// TIA Portal V16 export
// export: Created 2021-11-12T13:32:07.3551266Z, ExportSetting WithDefaults, DisplayName Totally Integrated Automation Portal, DisplayVersion V16 Update 3, DisplayName TIA Portal Version Control Interface, DisplayVersion V16 Update 2, DisplayName TIA Portal Openness, DisplayVersion V16 Update 3, DisplayName SINAMICS Startdrive Advanced, DisplayVersion V16 Update 5, DisplayName SINAMICS Startdrive G130, G150, S120, S150, SINAMICS MV, S210, DisplayVersion V16 Update 5, DisplayName SINAMICS Startdrive G110M, G120, G120C, G120D, G120P, G115D, DisplayVersion V16 Update 5, DisplayName STEP 7 Professional, DisplayVersion V16 Update 3, DisplayName STEP 7 Safety, DisplayVersion V16, DisplayName WinCC UA Professional, DisplayVersion V16 Update 3
FUNCTION_BLOCK "Station130"   // FB11, LAD
{ S7_Optimized_Access := 'TRUE' }
VERSION : 0.1
// stored: AutoNumber true, IsIECCheckEnabled false, IsRetainMemResEnabled false, MemoryReserve 100, SetENOAutomatically false, UDAEnableTagReadback false
   VAR
      SS_RobotZones : "STD_RobotZones";
      SI_PartType { S7_SetPoint := 'True'} : Int;
      SDI_PartID : DInt;
      SI_PartCounter : Int;
   END_VAR
   VAR_TEMP   // added for the SCL form of the ladder/FBD networks
      _w1 : Bool;
      _w2 : Bool;
      _w3 : Bool;
      _w4 : Bool;
      _w5 : Bool;
      _w6 : Bool;
      _w7 : Bool;
      _w8 : Bool;
      _w9 : Bool;
      _w10 : Bool;
      _w11 : Bool;
      _w12 : Bool;
      _w13 : Bool;
      _w14 : Bool;
      _w15 : Bool;
      _w16 : Bool;
      _w17 : Bool;
      _w18 : Bool;
      _w19 : Bool;
      _w20 : Bool;
      _w21 : Bool;
      _w22 : Bool;
      _w23 : Bool;
      _w24 : Bool;
      _w25 : Bool;
   END_VAR
BEGIN

REGION Network 1: *************** Clear Temporary ***************
END_REGION

REGION Network 2: *************** Zone release *************
END_REGION

REGION Network 3: Enable for robots 1R1, 1R3 to enter zone 130
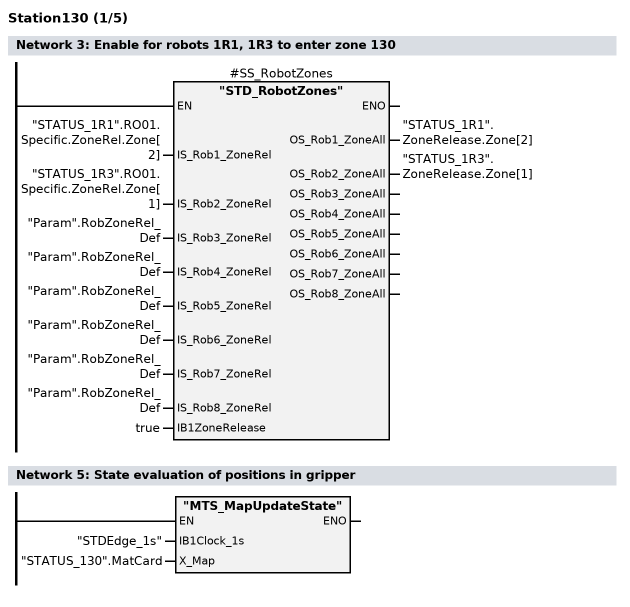
   RUNG wire#powerrail
      #SS_RobotZones(IS_Rob1_ZoneRel := "STATUS_1R1".RO01.Specific.ZoneRel.Zone[2], IS_Rob2_ZoneRel := "STATUS_1R3".RO01.Specific.ZoneRel.Zone[1], IS_Rob3_ZoneRel := "Param".RobZoneRel_Def, IS_Rob4_ZoneRel := "Param".RobZoneRel_Def, IS_Rob5_ZoneRel := "Param".RobZoneRel_Def, IS_Rob6_ZoneRel := "Param".RobZoneRel_Def, IS_Rob7_ZoneRel := "Param".RobZoneRel_Def, IS_Rob8_ZoneRel := "Param".RobZoneRel_Def, IB1ZoneRelease := true, OS_Rob1_ZoneAll => "STATUS_1R1".ZoneRelease.Zone[2], OS_Rob2_ZoneAll => "STATUS_1R3".ZoneRelease.Zone[1], OS_Rob3_ZoneAll =>, OS_Rob4_ZoneAll =>, OS_Rob5_ZoneAll =>, OS_Rob6_ZoneAll =>, OS_Rob7_ZoneAll =>, OS_Rob8_ZoneAll =>)
   END_RUNG
   // the same network as SCL:
   #SS_RobotZones(IS_Rob1_ZoneRel := "STATUS_1R1".RO01.Specific.ZoneRel.Zone[2],   // "STD_RobotZones"
                  IS_Rob2_ZoneRel := "STATUS_1R3".RO01.Specific.ZoneRel.Zone[1],
                  IS_Rob3_ZoneRel := "Param".RobZoneRel_Def,
                  IS_Rob4_ZoneRel := "Param".RobZoneRel_Def,
                  IS_Rob5_ZoneRel := "Param".RobZoneRel_Def,
                  IS_Rob6_ZoneRel := "Param".RobZoneRel_Def,
                  IS_Rob7_ZoneRel := "Param".RobZoneRel_Def,
                  IS_Rob8_ZoneRel := "Param".RobZoneRel_Def,
                  IB1ZoneRelease := true,
                  OS_Rob1_ZoneAll => "STATUS_1R1".ZoneRelease.Zone[2],
                  OS_Rob2_ZoneAll => "STATUS_1R3".ZoneRelease.Zone[1]);
END_REGION

REGION Network 4: *************** Material flow ***************
END_REGION

REGION Network 5: State evaluation of positions in gripper
   RUNG wire#powerrail
      "MTS_MapUpdateState"(IB1Clock_1s := "STDEdge_1s", X_Map := "STATUS_130".MatCard)
   END_RUNG
   // the same network as SCL:
   "MTS_MapUpdateState"(IB1Clock_1s := "STDEdge_1s", X_Map := "STATUS_130".MatCard);
END_REGION

REGION Network 6: Clear positions and map - commands
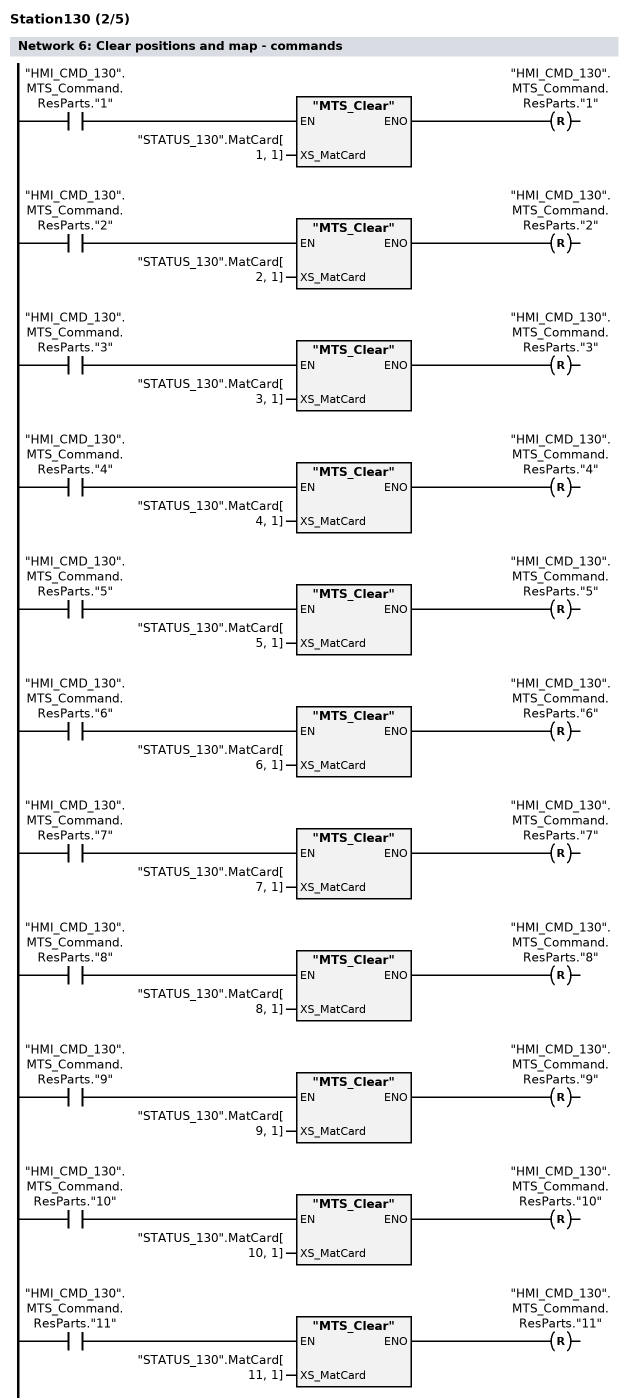
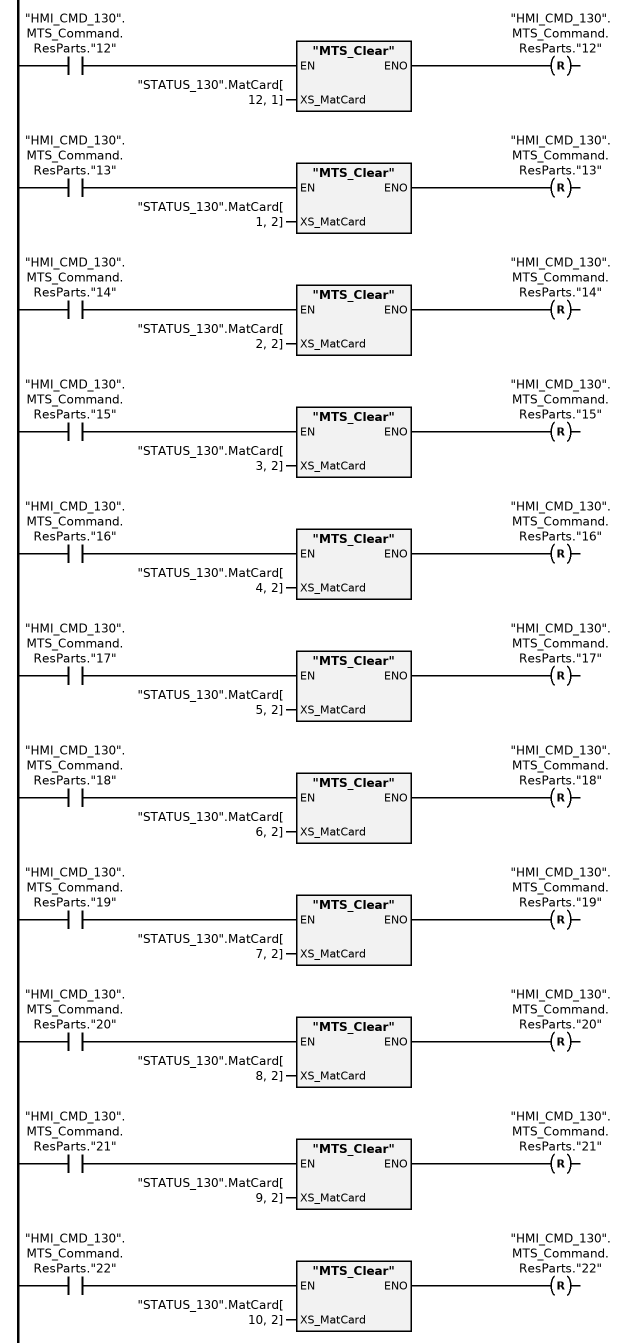
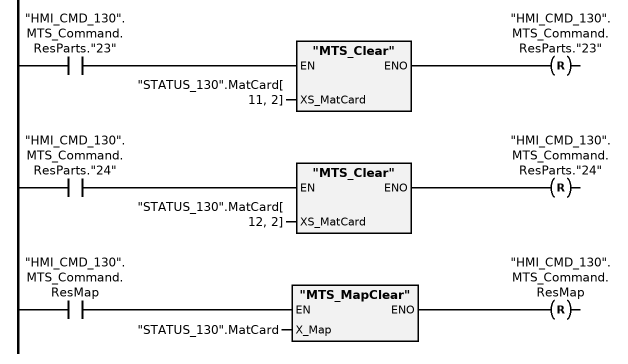
   RUNG wire#powerrail
      Contact( "HMI_CMD_130".MTS_Command.ResParts."1" )
      "MTS_Clear"(XS_MatCard := "STATUS_130".MatCard[1, 1])
      R_Coil( "HMI_CMD_130".MTS_Command.ResParts."1" )
   END_RUNG
   RUNG wire#powerrail
      Contact( "HMI_CMD_130".MTS_Command.ResParts."2" )
      "MTS_Clear"(XS_MatCard := "STATUS_130".MatCard[2, 1])
      R_Coil( "HMI_CMD_130".MTS_Command.ResParts."2" )
   END_RUNG
   RUNG wire#powerrail
      Contact( "HMI_CMD_130".MTS_Command.ResParts."3" )
      "MTS_Clear"(XS_MatCard := "STATUS_130".MatCard[3, 1])
      R_Coil( "HMI_CMD_130".MTS_Command.ResParts."3" )
   END_RUNG
   RUNG wire#powerrail
      Contact( "HMI_CMD_130".MTS_Command.ResParts."4" )
      "MTS_Clear"(XS_MatCard := "STATUS_130".MatCard[4, 1])
      R_Coil( "HMI_CMD_130".MTS_Command.ResParts."4" )
   END_RUNG
   RUNG wire#powerrail
      Contact( "HMI_CMD_130".MTS_Command.ResParts."5" )
      "MTS_Clear"(XS_MatCard := "STATUS_130".MatCard[5, 1])
      R_Coil( "HMI_CMD_130".MTS_Command.ResParts."5" )
   END_RUNG
   RUNG wire#powerrail
      Contact( "HMI_CMD_130".MTS_Command.ResParts."6" )
      "MTS_Clear"(XS_MatCard := "STATUS_130".MatCard[6, 1])
      R_Coil( "HMI_CMD_130".MTS_Command.ResParts."6" )
   END_RUNG
   RUNG wire#powerrail
      Contact( "HMI_CMD_130".MTS_Command.ResParts."7" )
      "MTS_Clear"(XS_MatCard := "STATUS_130".MatCard[7, 1])
      R_Coil( "HMI_CMD_130".MTS_Command.ResParts."7" )
   END_RUNG
   RUNG wire#powerrail
      Contact( "HMI_CMD_130".MTS_Command.ResParts."8" )
      "MTS_Clear"(XS_MatCard := "STATUS_130".MatCard[8, 1])
      R_Coil( "HMI_CMD_130".MTS_Command.ResParts."8" )
   END_RUNG
   RUNG wire#powerrail
      Contact( "HMI_CMD_130".MTS_Command.ResParts."9" )
      "MTS_Clear"(XS_MatCard := "STATUS_130".MatCard[9, 1])
      R_Coil( "HMI_CMD_130".MTS_Command.ResParts."9" )
   END_RUNG
   RUNG wire#powerrail
      Contact( "HMI_CMD_130".MTS_Command.ResParts."10" )
      "MTS_Clear"(XS_MatCard := "STATUS_130".MatCard[10, 1])
      R_Coil( "HMI_CMD_130".MTS_Command.ResParts."10" )
   END_RUNG
   RUNG wire#powerrail
      Contact( "HMI_CMD_130".MTS_Command.ResParts."11" )
      "MTS_Clear"(XS_MatCard := "STATUS_130".MatCard[11, 1])
      R_Coil( "HMI_CMD_130".MTS_Command.ResParts."11" )
   END_RUNG
   RUNG wire#powerrail
      Contact( "HMI_CMD_130".MTS_Command.ResParts."12" )
      "MTS_Clear"(XS_MatCard := "STATUS_130".MatCard[12, 1])
      R_Coil( "HMI_CMD_130".MTS_Command.ResParts."12" )
   END_RUNG
   RUNG wire#powerrail
      Contact( "HMI_CMD_130".MTS_Command.ResParts."13" )
      "MTS_Clear"(XS_MatCard := "STATUS_130".MatCard[1, 2])
      R_Coil( "HMI_CMD_130".MTS_Command.ResParts."13" )
   END_RUNG
   RUNG wire#powerrail
      Contact( "HMI_CMD_130".MTS_Command.ResParts."14" )
      "MTS_Clear"(XS_MatCard := "STATUS_130".MatCard[2, 2])
      R_Coil( "HMI_CMD_130".MTS_Command.ResParts."14" )
   END_RUNG
   RUNG wire#powerrail
      Contact( "HMI_CMD_130".MTS_Command.ResParts."15" )
      "MTS_Clear"(XS_MatCard := "STATUS_130".MatCard[3, 2])
      R_Coil( "HMI_CMD_130".MTS_Command.ResParts."15" )
   END_RUNG
   RUNG wire#powerrail
      Contact( "HMI_CMD_130".MTS_Command.ResParts."16" )
      "MTS_Clear"(XS_MatCard := "STATUS_130".MatCard[4, 2])
      R_Coil( "HMI_CMD_130".MTS_Command.ResParts."16" )
   END_RUNG
   RUNG wire#powerrail
      Contact( "HMI_CMD_130".MTS_Command.ResParts."17" )
      "MTS_Clear"(XS_MatCard := "STATUS_130".MatCard[5, 2])
      R_Coil( "HMI_CMD_130".MTS_Command.ResParts."17" )
   END_RUNG
   RUNG wire#powerrail
      Contact( "HMI_CMD_130".MTS_Command.ResParts."18" )
      "MTS_Clear"(XS_MatCard := "STATUS_130".MatCard[6, 2])
      R_Coil( "HMI_CMD_130".MTS_Command.ResParts."18" )
   END_RUNG
   RUNG wire#powerrail
      Contact( "HMI_CMD_130".MTS_Command.ResParts."19" )
      "MTS_Clear"(XS_MatCard := "STATUS_130".MatCard[7, 2])
      R_Coil( "HMI_CMD_130".MTS_Command.ResParts."19" )
   END_RUNG
   RUNG wire#powerrail
      Contact( "HMI_CMD_130".MTS_Command.ResParts."20" )
      "MTS_Clear"(XS_MatCard := "STATUS_130".MatCard[8, 2])
      R_Coil( "HMI_CMD_130".MTS_Command.ResParts."20" )
   END_RUNG
   RUNG wire#powerrail
      Contact( "HMI_CMD_130".MTS_Command.ResParts."21" )
      "MTS_Clear"(XS_MatCard := "STATUS_130".MatCard[9, 2])
      R_Coil( "HMI_CMD_130".MTS_Command.ResParts."21" )
   END_RUNG
   RUNG wire#powerrail
      Contact( "HMI_CMD_130".MTS_Command.ResParts."22" )
      "MTS_Clear"(XS_MatCard := "STATUS_130".MatCard[10, 2])
      R_Coil( "HMI_CMD_130".MTS_Command.ResParts."22" )
   END_RUNG
   RUNG wire#powerrail
      Contact( "HMI_CMD_130".MTS_Command.ResParts."23" )
      "MTS_Clear"(XS_MatCard := "STATUS_130".MatCard[11, 2])
      R_Coil( "HMI_CMD_130".MTS_Command.ResParts."23" )
   END_RUNG
   RUNG wire#powerrail
      Contact( "HMI_CMD_130".MTS_Command.ResParts."24" )
      "MTS_Clear"(XS_MatCard := "STATUS_130".MatCard[12, 2])
      R_Coil( "HMI_CMD_130".MTS_Command.ResParts."24" )
   END_RUNG
   RUNG wire#powerrail
      Contact( "HMI_CMD_130".MTS_Command.ResMap )
      "MTS_MapClear"(X_Map := "STATUS_130".MatCard)
      R_Coil( "HMI_CMD_130".MTS_Command.ResMap )
   END_RUNG
   // the same network as SCL:
   "MTS_Clear"(EN := "HMI_CMD_130".MTS_Command.ResParts."1",
               XS_MatCard := "STATUS_130".MatCard[1, 1],
               ENO => #_w1);
   IF #_w1 THEN "HMI_CMD_130".MTS_Command.ResParts."1" := FALSE; END_IF;
   "MTS_Clear"(EN := "HMI_CMD_130".MTS_Command.ResParts."2",
               XS_MatCard := "STATUS_130".MatCard[2, 1],
               ENO => #_w2);
   IF #_w2 THEN "HMI_CMD_130".MTS_Command.ResParts."2" := FALSE; END_IF;
   "MTS_Clear"(EN := "HMI_CMD_130".MTS_Command.ResParts."3",
               XS_MatCard := "STATUS_130".MatCard[3, 1],
               ENO => #_w3);
   IF #_w3 THEN "HMI_CMD_130".MTS_Command.ResParts."3" := FALSE; END_IF;
   "MTS_Clear"(EN := "HMI_CMD_130".MTS_Command.ResParts."4",
               XS_MatCard := "STATUS_130".MatCard[4, 1],
               ENO => #_w4);
   IF #_w4 THEN "HMI_CMD_130".MTS_Command.ResParts."4" := FALSE; END_IF;
   "MTS_Clear"(EN := "HMI_CMD_130".MTS_Command.ResParts."5",
               XS_MatCard := "STATUS_130".MatCard[5, 1],
               ENO => #_w5);
   IF #_w5 THEN "HMI_CMD_130".MTS_Command.ResParts."5" := FALSE; END_IF;
   "MTS_Clear"(EN := "HMI_CMD_130".MTS_Command.ResParts."6",
               XS_MatCard := "STATUS_130".MatCard[6, 1],
               ENO => #_w6);
   IF #_w6 THEN "HMI_CMD_130".MTS_Command.ResParts."6" := FALSE; END_IF;
   "MTS_Clear"(EN := "HMI_CMD_130".MTS_Command.ResParts."7",
               XS_MatCard := "STATUS_130".MatCard[7, 1],
               ENO => #_w7);
   IF #_w7 THEN "HMI_CMD_130".MTS_Command.ResParts."7" := FALSE; END_IF;
   "MTS_Clear"(EN := "HMI_CMD_130".MTS_Command.ResParts."8",
               XS_MatCard := "STATUS_130".MatCard[8, 1],
               ENO => #_w8);
   IF #_w8 THEN "HMI_CMD_130".MTS_Command.ResParts."8" := FALSE; END_IF;
   "MTS_Clear"(EN := "HMI_CMD_130".MTS_Command.ResParts."9",
               XS_MatCard := "STATUS_130".MatCard[9, 1],
               ENO => #_w9);
   IF #_w9 THEN "HMI_CMD_130".MTS_Command.ResParts."9" := FALSE; END_IF;
   "MTS_Clear"(EN := "HMI_CMD_130".MTS_Command.ResParts."10",
               XS_MatCard := "STATUS_130".MatCard[10, 1],
               ENO => #_w10);
   IF #_w10 THEN "HMI_CMD_130".MTS_Command.ResParts."10" := FALSE; END_IF;
   "MTS_Clear"(EN := "HMI_CMD_130".MTS_Command.ResParts."11",
               XS_MatCard := "STATUS_130".MatCard[11, 1],
               ENO => #_w11);
   IF #_w11 THEN "HMI_CMD_130".MTS_Command.ResParts."11" := FALSE; END_IF;
   "MTS_Clear"(EN := "HMI_CMD_130".MTS_Command.ResParts."12",
               XS_MatCard := "STATUS_130".MatCard[12, 1],
               ENO => #_w12);
   IF #_w12 THEN "HMI_CMD_130".MTS_Command.ResParts."12" := FALSE; END_IF;
   "MTS_Clear"(EN := "HMI_CMD_130".MTS_Command.ResParts."13",
               XS_MatCard := "STATUS_130".MatCard[1, 2],
               ENO => #_w13);
   IF #_w13 THEN "HMI_CMD_130".MTS_Command.ResParts."13" := FALSE; END_IF;
   "MTS_Clear"(EN := "HMI_CMD_130".MTS_Command.ResParts."14",
               XS_MatCard := "STATUS_130".MatCard[2, 2],
               ENO => #_w14);
   IF #_w14 THEN "HMI_CMD_130".MTS_Command.ResParts."14" := FALSE; END_IF;
   "MTS_Clear"(EN := "HMI_CMD_130".MTS_Command.ResParts."15",
               XS_MatCard := "STATUS_130".MatCard[3, 2],
               ENO => #_w15);
   IF #_w15 THEN "HMI_CMD_130".MTS_Command.ResParts."15" := FALSE; END_IF;
   "MTS_Clear"(EN := "HMI_CMD_130".MTS_Command.ResParts."16",
               XS_MatCard := "STATUS_130".MatCard[4, 2],
               ENO => #_w16);
   IF #_w16 THEN "HMI_CMD_130".MTS_Command.ResParts."16" := FALSE; END_IF;
   "MTS_Clear"(EN := "HMI_CMD_130".MTS_Command.ResParts."17",
               XS_MatCard := "STATUS_130".MatCard[5, 2],
               ENO => #_w17);
   IF #_w17 THEN "HMI_CMD_130".MTS_Command.ResParts."17" := FALSE; END_IF;
   "MTS_Clear"(EN := "HMI_CMD_130".MTS_Command.ResParts."18",
               XS_MatCard := "STATUS_130".MatCard[6, 2],
               ENO => #_w18);
   IF #_w18 THEN "HMI_CMD_130".MTS_Command.ResParts."18" := FALSE; END_IF;
   "MTS_Clear"(EN := "HMI_CMD_130".MTS_Command.ResParts."19",
               XS_MatCard := "STATUS_130".MatCard[7, 2],
               ENO => #_w19);
   IF #_w19 THEN "HMI_CMD_130".MTS_Command.ResParts."19" := FALSE; END_IF;
   "MTS_Clear"(EN := "HMI_CMD_130".MTS_Command.ResParts."20",
               XS_MatCard := "STATUS_130".MatCard[8, 2],
               ENO => #_w20);
   IF #_w20 THEN "HMI_CMD_130".MTS_Command.ResParts."20" := FALSE; END_IF;
   "MTS_Clear"(EN := "HMI_CMD_130".MTS_Command.ResParts."21",
               XS_MatCard := "STATUS_130".MatCard[9, 2],
               ENO => #_w21);
   IF #_w21 THEN "HMI_CMD_130".MTS_Command.ResParts."21" := FALSE; END_IF;
   "MTS_Clear"(EN := "HMI_CMD_130".MTS_Command.ResParts."22",
               XS_MatCard := "STATUS_130".MatCard[10, 2],
               ENO => #_w22);
   IF #_w22 THEN "HMI_CMD_130".MTS_Command.ResParts."22" := FALSE; END_IF;
   "MTS_Clear"(EN := "HMI_CMD_130".MTS_Command.ResParts."23",
               XS_MatCard := "STATUS_130".MatCard[11, 2],
               ENO => #_w23);
   IF #_w23 THEN "HMI_CMD_130".MTS_Command.ResParts."23" := FALSE; END_IF;
   "MTS_Clear"(EN := "HMI_CMD_130".MTS_Command.ResParts."24",
               XS_MatCard := "STATUS_130".MatCard[12, 2],
               ENO => #_w24);
   IF #_w24 THEN "HMI_CMD_130".MTS_Command.ResParts."24" := FALSE; END_IF;
   "MTS_MapClear"(EN := "HMI_CMD_130".MTS_Command.ResMap, X_Map := "STATUS_130".MatCard, ENO => #_w25);
   IF #_w25 THEN "HMI_CMD_130".MTS_Command.ResMap := FALSE; END_IF;
END_REGION

REGION Network 7: Set positions - init
   // "JSA0Comm" - change when recipes done
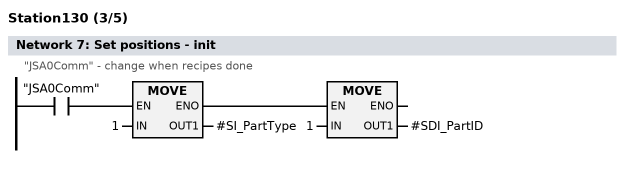
   RUNG wire#powerrail
      Contact( "JSA0Comm" )
      Move(in := 1, out1 => #SI_PartType)
      Move(in := 1, out1 => #SDI_PartID)
   END_RUNG
   // the same network as SCL:
   IF "JSA0Comm" THEN
       #SI_PartType := 1;
       #SDI_PartID := 1;
   END_IF;
END_REGION

REGION Network 8: Set positions and map - commands
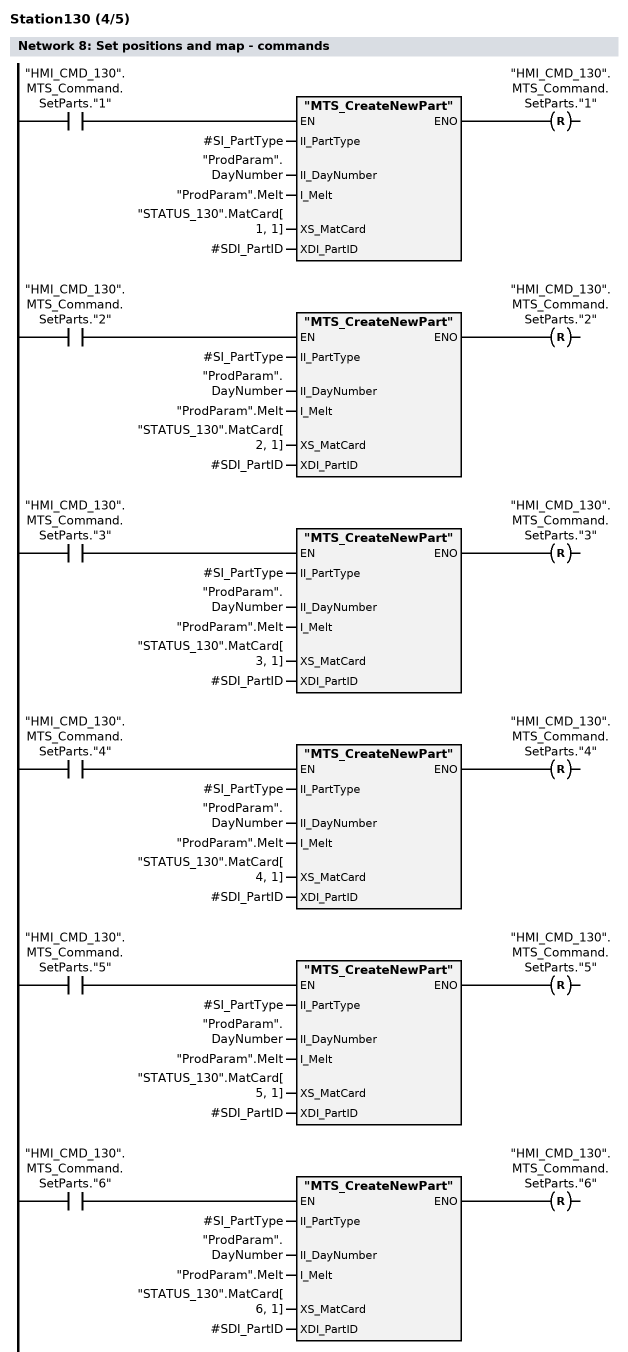
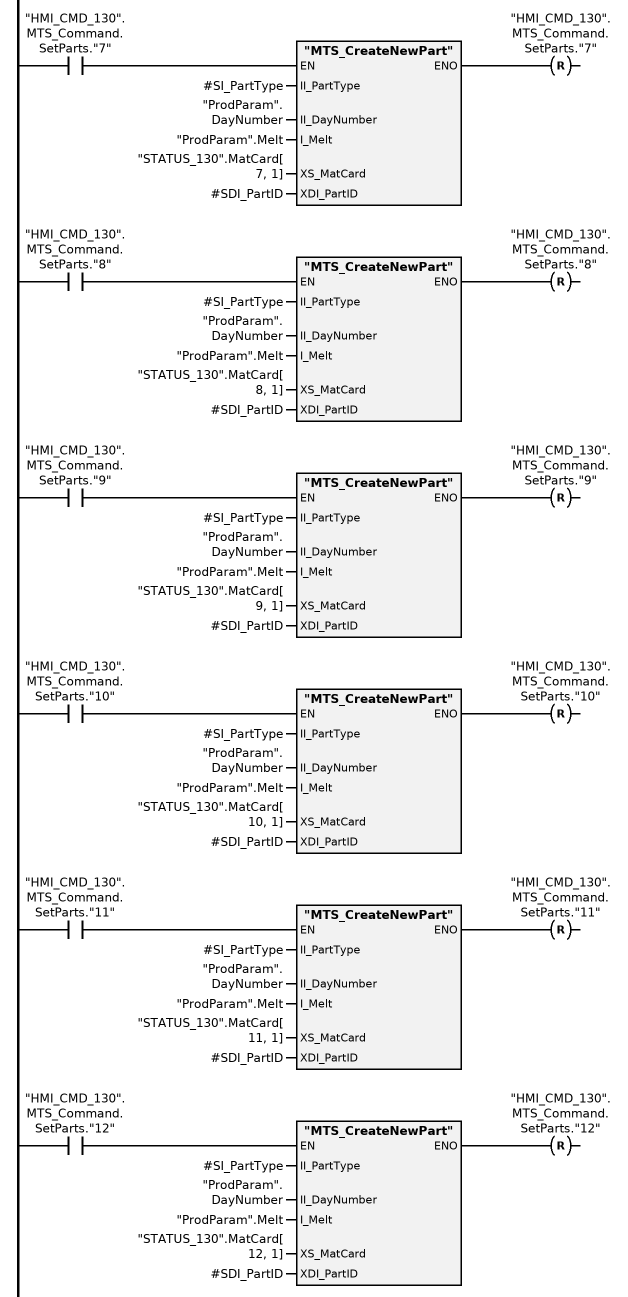
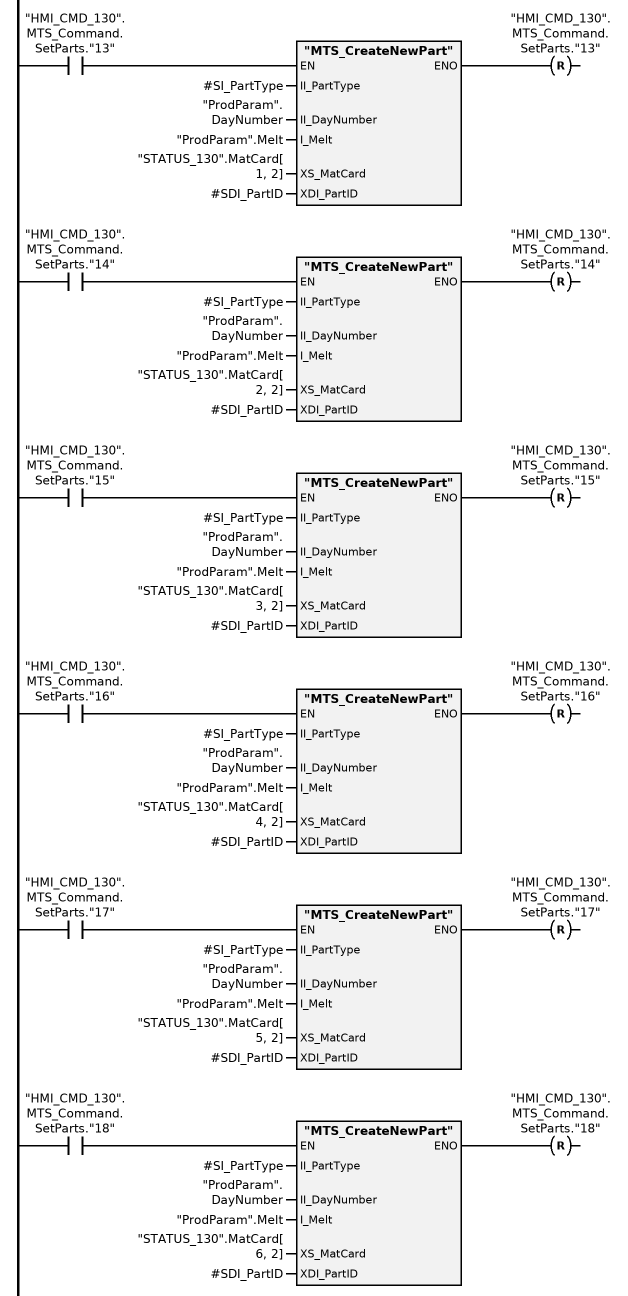
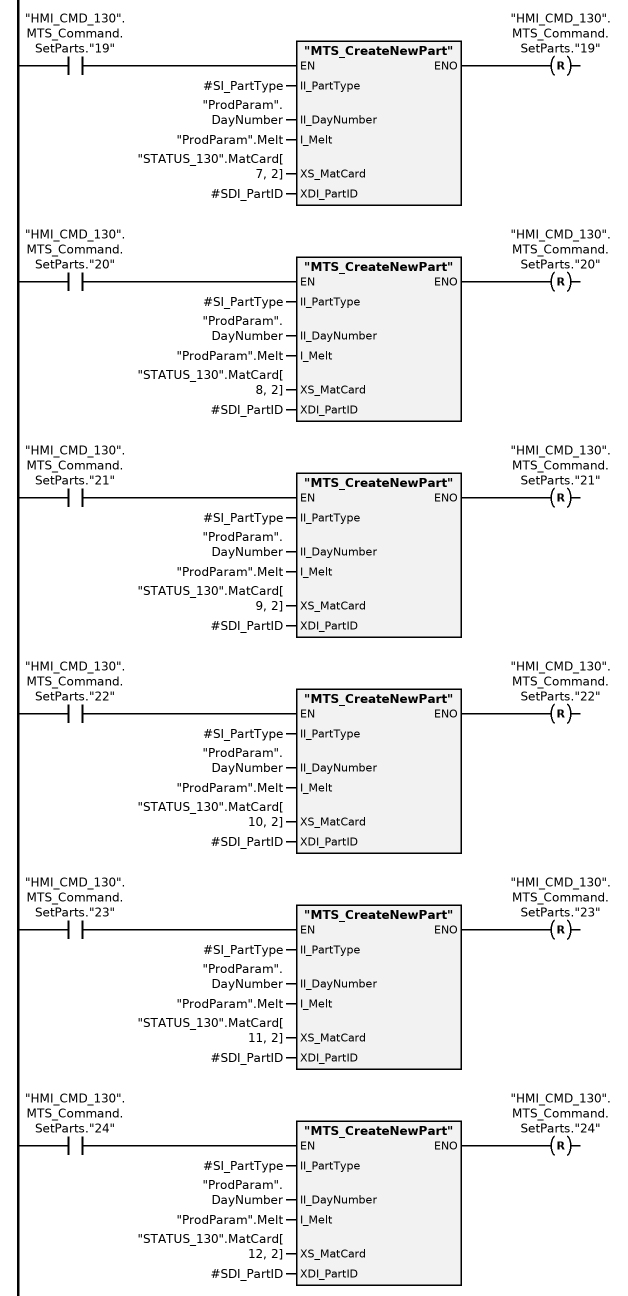
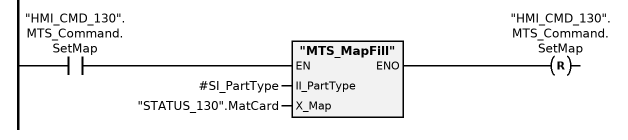
   RUNG wire#powerrail
      Contact( "HMI_CMD_130".MTS_Command.SetParts."1" )
      "MTS_CreateNewPart"(II_PartType := #SI_PartType, II_DayNumber := "ProdParam".DayNumber, I_Melt := "ProdParam".Melt, XS_MatCard := "STATUS_130".MatCard[1, 1], XDI_PartID := #SDI_PartID)
      R_Coil( "HMI_CMD_130".MTS_Command.SetParts."1" )
   END_RUNG
   RUNG wire#powerrail
      Contact( "HMI_CMD_130".MTS_Command.SetParts."2" )
      "MTS_CreateNewPart"(II_PartType := #SI_PartType, II_DayNumber := "ProdParam".DayNumber, I_Melt := "ProdParam".Melt, XS_MatCard := "STATUS_130".MatCard[2, 1], XDI_PartID := #SDI_PartID)
      R_Coil( "HMI_CMD_130".MTS_Command.SetParts."2" )
   END_RUNG
   RUNG wire#powerrail
      Contact( "HMI_CMD_130".MTS_Command.SetParts."3" )
      "MTS_CreateNewPart"(II_PartType := #SI_PartType, II_DayNumber := "ProdParam".DayNumber, I_Melt := "ProdParam".Melt, XS_MatCard := "STATUS_130".MatCard[3, 1], XDI_PartID := #SDI_PartID)
      R_Coil( "HMI_CMD_130".MTS_Command.SetParts."3" )
   END_RUNG
   RUNG wire#powerrail
      Contact( "HMI_CMD_130".MTS_Command.SetParts."4" )
      "MTS_CreateNewPart"(II_PartType := #SI_PartType, II_DayNumber := "ProdParam".DayNumber, I_Melt := "ProdParam".Melt, XS_MatCard := "STATUS_130".MatCard[4, 1], XDI_PartID := #SDI_PartID)
      R_Coil( "HMI_CMD_130".MTS_Command.SetParts."4" )
   END_RUNG
   RUNG wire#powerrail
      Contact( "HMI_CMD_130".MTS_Command.SetParts."5" )
      "MTS_CreateNewPart"(II_PartType := #SI_PartType, II_DayNumber := "ProdParam".DayNumber, I_Melt := "ProdParam".Melt, XS_MatCard := "STATUS_130".MatCard[5, 1], XDI_PartID := #SDI_PartID)
      R_Coil( "HMI_CMD_130".MTS_Command.SetParts."5" )
   END_RUNG
   RUNG wire#powerrail
      Contact( "HMI_CMD_130".MTS_Command.SetParts."6" )
      "MTS_CreateNewPart"(II_PartType := #SI_PartType, II_DayNumber := "ProdParam".DayNumber, I_Melt := "ProdParam".Melt, XS_MatCard := "STATUS_130".MatCard[6, 1], XDI_PartID := #SDI_PartID)
      R_Coil( "HMI_CMD_130".MTS_Command.SetParts."6" )
   END_RUNG
   RUNG wire#powerrail
      Contact( "HMI_CMD_130".MTS_Command.SetParts."7" )
      "MTS_CreateNewPart"(II_PartType := #SI_PartType, II_DayNumber := "ProdParam".DayNumber, I_Melt := "ProdParam".Melt, XS_MatCard := "STATUS_130".MatCard[7, 1], XDI_PartID := #SDI_PartID)
      R_Coil( "HMI_CMD_130".MTS_Command.SetParts."7" )
   END_RUNG
   RUNG wire#powerrail
      Contact( "HMI_CMD_130".MTS_Command.SetParts."8" )
      "MTS_CreateNewPart"(II_PartType := #SI_PartType, II_DayNumber := "ProdParam".DayNumber, I_Melt := "ProdParam".Melt, XS_MatCard := "STATUS_130".MatCard[8, 1], XDI_PartID := #SDI_PartID)
      R_Coil( "HMI_CMD_130".MTS_Command.SetParts."8" )
   END_RUNG
   RUNG wire#powerrail
      Contact( "HMI_CMD_130".MTS_Command.SetParts."9" )
      "MTS_CreateNewPart"(II_PartType := #SI_PartType, II_DayNumber := "ProdParam".DayNumber, I_Melt := "ProdParam".Melt, XS_MatCard := "STATUS_130".MatCard[9, 1], XDI_PartID := #SDI_PartID)
      R_Coil( "HMI_CMD_130".MTS_Command.SetParts."9" )
   END_RUNG
   RUNG wire#powerrail
      Contact( "HMI_CMD_130".MTS_Command.SetParts."10" )
      "MTS_CreateNewPart"(II_PartType := #SI_PartType, II_DayNumber := "ProdParam".DayNumber, I_Melt := "ProdParam".Melt, XS_MatCard := "STATUS_130".MatCard[10, 1], XDI_PartID := #SDI_PartID)
      R_Coil( "HMI_CMD_130".MTS_Command.SetParts."10" )
   END_RUNG
   RUNG wire#powerrail
      Contact( "HMI_CMD_130".MTS_Command.SetParts."11" )
      "MTS_CreateNewPart"(II_PartType := #SI_PartType, II_DayNumber := "ProdParam".DayNumber, I_Melt := "ProdParam".Melt, XS_MatCard := "STATUS_130".MatCard[11, 1], XDI_PartID := #SDI_PartID)
      R_Coil( "HMI_CMD_130".MTS_Command.SetParts."11" )
   END_RUNG
   RUNG wire#powerrail
      Contact( "HMI_CMD_130".MTS_Command.SetParts."12" )
      "MTS_CreateNewPart"(II_PartType := #SI_PartType, II_DayNumber := "ProdParam".DayNumber, I_Melt := "ProdParam".Melt, XS_MatCard := "STATUS_130".MatCard[12, 1], XDI_PartID := #SDI_PartID)
      R_Coil( "HMI_CMD_130".MTS_Command.SetParts."12" )
   END_RUNG
   RUNG wire#powerrail
      Contact( "HMI_CMD_130".MTS_Command.SetParts."13" )
      "MTS_CreateNewPart"(II_PartType := #SI_PartType, II_DayNumber := "ProdParam".DayNumber, I_Melt := "ProdParam".Melt, XS_MatCard := "STATUS_130".MatCard[1, 2], XDI_PartID := #SDI_PartID)
      R_Coil( "HMI_CMD_130".MTS_Command.SetParts."13" )
   END_RUNG
   RUNG wire#powerrail
      Contact( "HMI_CMD_130".MTS_Command.SetParts."14" )
      "MTS_CreateNewPart"(II_PartType := #SI_PartType, II_DayNumber := "ProdParam".DayNumber, I_Melt := "ProdParam".Melt, XS_MatCard := "STATUS_130".MatCard[2, 2], XDI_PartID := #SDI_PartID)
      R_Coil( "HMI_CMD_130".MTS_Command.SetParts."14" )
   END_RUNG
   RUNG wire#powerrail
      Contact( "HMI_CMD_130".MTS_Command.SetParts."15" )
      "MTS_CreateNewPart"(II_PartType := #SI_PartType, II_DayNumber := "ProdParam".DayNumber, I_Melt := "ProdParam".Melt, XS_MatCard := "STATUS_130".MatCard[3, 2], XDI_PartID := #SDI_PartID)
      R_Coil( "HMI_CMD_130".MTS_Command.SetParts."15" )
   END_RUNG
   RUNG wire#powerrail
      Contact( "HMI_CMD_130".MTS_Command.SetParts."16" )
      "MTS_CreateNewPart"(II_PartType := #SI_PartType, II_DayNumber := "ProdParam".DayNumber, I_Melt := "ProdParam".Melt, XS_MatCard := "STATUS_130".MatCard[4, 2], XDI_PartID := #SDI_PartID)
      R_Coil( "HMI_CMD_130".MTS_Command.SetParts."16" )
   END_RUNG
   RUNG wire#powerrail
      Contact( "HMI_CMD_130".MTS_Command.SetParts."17" )
      "MTS_CreateNewPart"(II_PartType := #SI_PartType, II_DayNumber := "ProdParam".DayNumber, I_Melt := "ProdParam".Melt, XS_MatCard := "STATUS_130".MatCard[5, 2], XDI_PartID := #SDI_PartID)
      R_Coil( "HMI_CMD_130".MTS_Command.SetParts."17" )
   END_RUNG
   RUNG wire#powerrail
      Contact( "HMI_CMD_130".MTS_Command.SetParts."18" )
      "MTS_CreateNewPart"(II_PartType := #SI_PartType, II_DayNumber := "ProdParam".DayNumber, I_Melt := "ProdParam".Melt, XS_MatCard := "STATUS_130".MatCard[6, 2], XDI_PartID := #SDI_PartID)
      R_Coil( "HMI_CMD_130".MTS_Command.SetParts."18" )
   END_RUNG
   RUNG wire#powerrail
      Contact( "HMI_CMD_130".MTS_Command.SetParts."19" )
      "MTS_CreateNewPart"(II_PartType := #SI_PartType, II_DayNumber := "ProdParam".DayNumber, I_Melt := "ProdParam".Melt, XS_MatCard := "STATUS_130".MatCard[7, 2], XDI_PartID := #SDI_PartID)
      R_Coil( "HMI_CMD_130".MTS_Command.SetParts."19" )
   END_RUNG
   RUNG wire#powerrail
      Contact( "HMI_CMD_130".MTS_Command.SetParts."20" )
      "MTS_CreateNewPart"(II_PartType := #SI_PartType, II_DayNumber := "ProdParam".DayNumber, I_Melt := "ProdParam".Melt, XS_MatCard := "STATUS_130".MatCard[8, 2], XDI_PartID := #SDI_PartID)
      R_Coil( "HMI_CMD_130".MTS_Command.SetParts."20" )
   END_RUNG
   RUNG wire#powerrail
      Contact( "HMI_CMD_130".MTS_Command.SetParts."21" )
      "MTS_CreateNewPart"(II_PartType := #SI_PartType, II_DayNumber := "ProdParam".DayNumber, I_Melt := "ProdParam".Melt, XS_MatCard := "STATUS_130".MatCard[9, 2], XDI_PartID := #SDI_PartID)
      R_Coil( "HMI_CMD_130".MTS_Command.SetParts."21" )
   END_RUNG
   RUNG wire#powerrail
      Contact( "HMI_CMD_130".MTS_Command.SetParts."22" )
      "MTS_CreateNewPart"(II_PartType := #SI_PartType, II_DayNumber := "ProdParam".DayNumber, I_Melt := "ProdParam".Melt, XS_MatCard := "STATUS_130".MatCard[10, 2], XDI_PartID := #SDI_PartID)
      R_Coil( "HMI_CMD_130".MTS_Command.SetParts."22" )
   END_RUNG
   RUNG wire#powerrail
      Contact( "HMI_CMD_130".MTS_Command.SetParts."23" )
      "MTS_CreateNewPart"(II_PartType := #SI_PartType, II_DayNumber := "ProdParam".DayNumber, I_Melt := "ProdParam".Melt, XS_MatCard := "STATUS_130".MatCard[11, 2], XDI_PartID := #SDI_PartID)
      R_Coil( "HMI_CMD_130".MTS_Command.SetParts."23" )
   END_RUNG
   RUNG wire#powerrail
      Contact( "HMI_CMD_130".MTS_Command.SetParts."24" )
      "MTS_CreateNewPart"(II_PartType := #SI_PartType, II_DayNumber := "ProdParam".DayNumber, I_Melt := "ProdParam".Melt, XS_MatCard := "STATUS_130".MatCard[12, 2], XDI_PartID := #SDI_PartID)
      R_Coil( "HMI_CMD_130".MTS_Command.SetParts."24" )
   END_RUNG
   RUNG wire#powerrail
      Contact( "HMI_CMD_130".MTS_Command.SetMap )
      "MTS_MapFill"(II_PartType := #SI_PartType, X_Map := "STATUS_130".MatCard)
      R_Coil( "HMI_CMD_130".MTS_Command.SetMap )
   END_RUNG
   // the same network as SCL:
   "MTS_CreateNewPart"(EN := "HMI_CMD_130".MTS_Command.SetParts."1",
                       II_PartType := #SI_PartType,
                       II_DayNumber := "ProdParam".DayNumber,
                       I_Melt := "ProdParam".Melt,
                       XS_MatCard := "STATUS_130".MatCard[1, 1],
                       XDI_PartID := #SDI_PartID,
                       ENO => #_w1);
   IF #_w1 THEN "HMI_CMD_130".MTS_Command.SetParts."1" := FALSE; END_IF;
   "MTS_CreateNewPart"(EN := "HMI_CMD_130".MTS_Command.SetParts."2",
                       II_PartType := #SI_PartType,
                       II_DayNumber := "ProdParam".DayNumber,
                       I_Melt := "ProdParam".Melt,
                       XS_MatCard := "STATUS_130".MatCard[2, 1],
                       XDI_PartID := #SDI_PartID,
                       ENO => #_w2);
   IF #_w2 THEN "HMI_CMD_130".MTS_Command.SetParts."2" := FALSE; END_IF;
   "MTS_CreateNewPart"(EN := "HMI_CMD_130".MTS_Command.SetParts."3",
                       II_PartType := #SI_PartType,
                       II_DayNumber := "ProdParam".DayNumber,
                       I_Melt := "ProdParam".Melt,
                       XS_MatCard := "STATUS_130".MatCard[3, 1],
                       XDI_PartID := #SDI_PartID,
                       ENO => #_w3);
   IF #_w3 THEN "HMI_CMD_130".MTS_Command.SetParts."3" := FALSE; END_IF;
   "MTS_CreateNewPart"(EN := "HMI_CMD_130".MTS_Command.SetParts."4",
                       II_PartType := #SI_PartType,
                       II_DayNumber := "ProdParam".DayNumber,
                       I_Melt := "ProdParam".Melt,
                       XS_MatCard := "STATUS_130".MatCard[4, 1],
                       XDI_PartID := #SDI_PartID,
                       ENO => #_w4);
   IF #_w4 THEN "HMI_CMD_130".MTS_Command.SetParts."4" := FALSE; END_IF;
   "MTS_CreateNewPart"(EN := "HMI_CMD_130".MTS_Command.SetParts."5",
                       II_PartType := #SI_PartType,
                       II_DayNumber := "ProdParam".DayNumber,
                       I_Melt := "ProdParam".Melt,
                       XS_MatCard := "STATUS_130".MatCard[5, 1],
                       XDI_PartID := #SDI_PartID,
                       ENO => #_w5);
   IF #_w5 THEN "HMI_CMD_130".MTS_Command.SetParts."5" := FALSE; END_IF;
   "MTS_CreateNewPart"(EN := "HMI_CMD_130".MTS_Command.SetParts."6",
                       II_PartType := #SI_PartType,
                       II_DayNumber := "ProdParam".DayNumber,
                       I_Melt := "ProdParam".Melt,
                       XS_MatCard := "STATUS_130".MatCard[6, 1],
                       XDI_PartID := #SDI_PartID,
                       ENO => #_w6);
   IF #_w6 THEN "HMI_CMD_130".MTS_Command.SetParts."6" := FALSE; END_IF;
   "MTS_CreateNewPart"(EN := "HMI_CMD_130".MTS_Command.SetParts."7",
                       II_PartType := #SI_PartType,
                       II_DayNumber := "ProdParam".DayNumber,
                       I_Melt := "ProdParam".Melt,
                       XS_MatCard := "STATUS_130".MatCard[7, 1],
                       XDI_PartID := #SDI_PartID,
                       ENO => #_w7);
   IF #_w7 THEN "HMI_CMD_130".MTS_Command.SetParts."7" := FALSE; END_IF;
   "MTS_CreateNewPart"(EN := "HMI_CMD_130".MTS_Command.SetParts."8",
                       II_PartType := #SI_PartType,
                       II_DayNumber := "ProdParam".DayNumber,
                       I_Melt := "ProdParam".Melt,
                       XS_MatCard := "STATUS_130".MatCard[8, 1],
                       XDI_PartID := #SDI_PartID,
                       ENO => #_w8);
   IF #_w8 THEN "HMI_CMD_130".MTS_Command.SetParts."8" := FALSE; END_IF;
   "MTS_CreateNewPart"(EN := "HMI_CMD_130".MTS_Command.SetParts."9",
                       II_PartType := #SI_PartType,
                       II_DayNumber := "ProdParam".DayNumber,
                       I_Melt := "ProdParam".Melt,
                       XS_MatCard := "STATUS_130".MatCard[9, 1],
                       XDI_PartID := #SDI_PartID,
                       ENO => #_w9);
   IF #_w9 THEN "HMI_CMD_130".MTS_Command.SetParts."9" := FALSE; END_IF;
   "MTS_CreateNewPart"(EN := "HMI_CMD_130".MTS_Command.SetParts."10",
                       II_PartType := #SI_PartType,
                       II_DayNumber := "ProdParam".DayNumber,
                       I_Melt := "ProdParam".Melt,
                       XS_MatCard := "STATUS_130".MatCard[10, 1],
                       XDI_PartID := #SDI_PartID,
                       ENO => #_w10);
   IF #_w10 THEN "HMI_CMD_130".MTS_Command.SetParts."10" := FALSE; END_IF;
   "MTS_CreateNewPart"(EN := "HMI_CMD_130".MTS_Command.SetParts."11",
                       II_PartType := #SI_PartType,
                       II_DayNumber := "ProdParam".DayNumber,
                       I_Melt := "ProdParam".Melt,
                       XS_MatCard := "STATUS_130".MatCard[11, 1],
                       XDI_PartID := #SDI_PartID,
                       ENO => #_w11);
   IF #_w11 THEN "HMI_CMD_130".MTS_Command.SetParts."11" := FALSE; END_IF;
   "MTS_CreateNewPart"(EN := "HMI_CMD_130".MTS_Command.SetParts."12",
                       II_PartType := #SI_PartType,
                       II_DayNumber := "ProdParam".DayNumber,
                       I_Melt := "ProdParam".Melt,
                       XS_MatCard := "STATUS_130".MatCard[12, 1],
                       XDI_PartID := #SDI_PartID,
                       ENO => #_w12);
   IF #_w12 THEN "HMI_CMD_130".MTS_Command.SetParts."12" := FALSE; END_IF;
   "MTS_CreateNewPart"(EN := "HMI_CMD_130".MTS_Command.SetParts."13",
                       II_PartType := #SI_PartType,
                       II_DayNumber := "ProdParam".DayNumber,
                       I_Melt := "ProdParam".Melt,
                       XS_MatCard := "STATUS_130".MatCard[1, 2],
                       XDI_PartID := #SDI_PartID,
                       ENO => #_w13);
   IF #_w13 THEN "HMI_CMD_130".MTS_Command.SetParts."13" := FALSE; END_IF;
   "MTS_CreateNewPart"(EN := "HMI_CMD_130".MTS_Command.SetParts."14",
                       II_PartType := #SI_PartType,
                       II_DayNumber := "ProdParam".DayNumber,
                       I_Melt := "ProdParam".Melt,
                       XS_MatCard := "STATUS_130".MatCard[2, 2],
                       XDI_PartID := #SDI_PartID,
                       ENO => #_w14);
   IF #_w14 THEN "HMI_CMD_130".MTS_Command.SetParts."14" := FALSE; END_IF;
   "MTS_CreateNewPart"(EN := "HMI_CMD_130".MTS_Command.SetParts."15",
                       II_PartType := #SI_PartType,
                       II_DayNumber := "ProdParam".DayNumber,
                       I_Melt := "ProdParam".Melt,
                       XS_MatCard := "STATUS_130".MatCard[3, 2],
                       XDI_PartID := #SDI_PartID,
                       ENO => #_w15);
   IF #_w15 THEN "HMI_CMD_130".MTS_Command.SetParts."15" := FALSE; END_IF;
   "MTS_CreateNewPart"(EN := "HMI_CMD_130".MTS_Command.SetParts."16",
                       II_PartType := #SI_PartType,
                       II_DayNumber := "ProdParam".DayNumber,
                       I_Melt := "ProdParam".Melt,
                       XS_MatCard := "STATUS_130".MatCard[4, 2],
                       XDI_PartID := #SDI_PartID,
                       ENO => #_w16);
   IF #_w16 THEN "HMI_CMD_130".MTS_Command.SetParts."16" := FALSE; END_IF;
   "MTS_CreateNewPart"(EN := "HMI_CMD_130".MTS_Command.SetParts."17",
                       II_PartType := #SI_PartType,
                       II_DayNumber := "ProdParam".DayNumber,
                       I_Melt := "ProdParam".Melt,
                       XS_MatCard := "STATUS_130".MatCard[5, 2],
                       XDI_PartID := #SDI_PartID,
                       ENO => #_w17);
   IF #_w17 THEN "HMI_CMD_130".MTS_Command.SetParts."17" := FALSE; END_IF;
   "MTS_CreateNewPart"(EN := "HMI_CMD_130".MTS_Command.SetParts."18",
                       II_PartType := #SI_PartType,
                       II_DayNumber := "ProdParam".DayNumber,
                       I_Melt := "ProdParam".Melt,
                       XS_MatCard := "STATUS_130".MatCard[6, 2],
                       XDI_PartID := #SDI_PartID,
                       ENO => #_w18);
   IF #_w18 THEN "HMI_CMD_130".MTS_Command.SetParts."18" := FALSE; END_IF;
   "MTS_CreateNewPart"(EN := "HMI_CMD_130".MTS_Command.SetParts."19",
                       II_PartType := #SI_PartType,
                       II_DayNumber := "ProdParam".DayNumber,
                       I_Melt := "ProdParam".Melt,
                       XS_MatCard := "STATUS_130".MatCard[7, 2],
                       XDI_PartID := #SDI_PartID,
                       ENO => #_w19);
   IF #_w19 THEN "HMI_CMD_130".MTS_Command.SetParts."19" := FALSE; END_IF;
   "MTS_CreateNewPart"(EN := "HMI_CMD_130".MTS_Command.SetParts."20",
                       II_PartType := #SI_PartType,
                       II_DayNumber := "ProdParam".DayNumber,
                       I_Melt := "ProdParam".Melt,
                       XS_MatCard := "STATUS_130".MatCard[8, 2],
                       XDI_PartID := #SDI_PartID,
                       ENO => #_w20);
   IF #_w20 THEN "HMI_CMD_130".MTS_Command.SetParts."20" := FALSE; END_IF;
   "MTS_CreateNewPart"(EN := "HMI_CMD_130".MTS_Command.SetParts."21",
                       II_PartType := #SI_PartType,
                       II_DayNumber := "ProdParam".DayNumber,
                       I_Melt := "ProdParam".Melt,
                       XS_MatCard := "STATUS_130".MatCard[9, 2],
                       XDI_PartID := #SDI_PartID,
                       ENO => #_w21);
   IF #_w21 THEN "HMI_CMD_130".MTS_Command.SetParts."21" := FALSE; END_IF;
   "MTS_CreateNewPart"(EN := "HMI_CMD_130".MTS_Command.SetParts."22",
                       II_PartType := #SI_PartType,
                       II_DayNumber := "ProdParam".DayNumber,
                       I_Melt := "ProdParam".Melt,
                       XS_MatCard := "STATUS_130".MatCard[10, 2],
                       XDI_PartID := #SDI_PartID,
                       ENO => #_w22);
   IF #_w22 THEN "HMI_CMD_130".MTS_Command.SetParts."22" := FALSE; END_IF;
   "MTS_CreateNewPart"(EN := "HMI_CMD_130".MTS_Command.SetParts."23",
                       II_PartType := #SI_PartType,
                       II_DayNumber := "ProdParam".DayNumber,
                       I_Melt := "ProdParam".Melt,
                       XS_MatCard := "STATUS_130".MatCard[11, 2],
                       XDI_PartID := #SDI_PartID,
                       ENO => #_w23);
   IF #_w23 THEN "HMI_CMD_130".MTS_Command.SetParts."23" := FALSE; END_IF;
   "MTS_CreateNewPart"(EN := "HMI_CMD_130".MTS_Command.SetParts."24",
                       II_PartType := #SI_PartType,
                       II_DayNumber := "ProdParam".DayNumber,
                       I_Melt := "ProdParam".Melt,
                       XS_MatCard := "STATUS_130".MatCard[12, 2],
                       XDI_PartID := #SDI_PartID,
                       ENO => #_w24);
   IF #_w24 THEN "HMI_CMD_130".MTS_Command.SetParts."24" := FALSE; END_IF;
   "MTS_MapFill"(EN := "HMI_CMD_130".MTS_Command.SetMap,
                 II_PartType := #SI_PartType,
                 X_Map := "STATUS_130".MatCard,
                 ENO => #_w25);
   IF #_w25 THEN "HMI_CMD_130".MTS_Command.SetMap := FALSE; END_IF;
END_REGION

REGION Network 9: *************** Part counter ***************
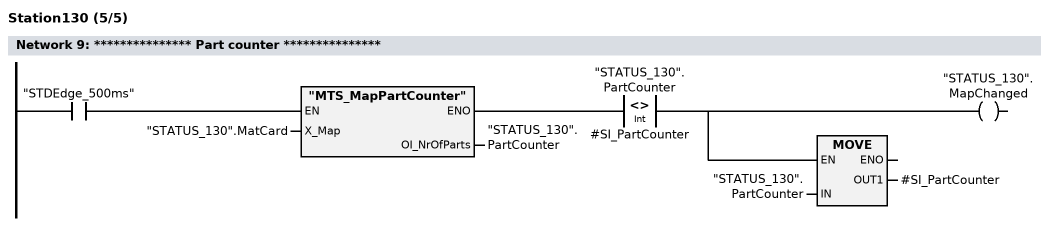
   RUNG wire#powerrail
      Contact( "STDEdge_500ms" )
      "MTS_MapPartCounter"(X_Map := "STATUS_130".MatCard, OI_NrOfParts => "STATUS_130".PartCounter)
      { S7_Templates := "SrcType := Int" } NE_Contact(in1 := "STATUS_130".PartCounter, in2 := #SI_PartCounter)
      wire#w1
      Coil( "STATUS_130".MapChanged )
   END_RUNG
   RUNG wire#w1
      Move(in := "STATUS_130".PartCounter, out1 => #SI_PartCounter)
   END_RUNG
   // the same network as SCL:
   "MTS_MapPartCounter"(EN := "STDEdge_500ms",
                        X_Map := "STATUS_130".MatCard,
                        OI_NrOfParts => "STATUS_130".PartCounter,
                        ENO => #_w1);
   "STATUS_130".MapChanged := #_w1 AND ("STATUS_130".PartCounter <> #SI_PartCounter);
   IF "STATUS_130".MapChanged THEN #SI_PartCounter := "STATUS_130".PartCounter; END_IF;
END_REGION
END_FUNCTION_BLOCK
